PROGRAM MAIN
VAR
	anchor : POINTER TO base;
	itf_anchor : POINTER TO ITF;
	
	parent : base;
	child1 : derived1;
	child2 : derived2;

	output : string;
END_VAR


anchor := ADR(parent);
output := anchor^.METH();

anchor := ADR(child1);
output := anchor^.METH();

anchor := ADR(child2);
output := anchor^.METH();
//polymorphism is possible

//complition error
itf_anchor := ADR(child1);
output := itf_anchor^.ITF_METH();

itf_anchor := ADR(child2);
output := itf_anchor^.ITF_METH();

END_PROGRAM

(* stored: Version 1.1.0.1, ProductVersion 3.1.4022.10
   POU MAIN: Id {3c7fcbe7-b0f5-4096-9e88-70b039acd9ca}, SpecialFunc None *)
